(* CODESYS project sfm MES Communication.project

Project tree, tasks and I/O mapping:
  Device : CODESYS Control for Raspberry Pi, 3S - Smart Software Solutions GmbH, version 3.5.11.20
    application Application
      libraries: Standard, * (System); Network, 3.5.7.0 (3S - Smart Software Solutions GmbH); Raspberry I2C Gyroscopes, 1.1.1.0 (3S - Smart Software Solutions GmbH)
      task MainTask (cyclic, interval 4 ms, priority 1) calls PLC_PRG
      task VISU_TASK (cyclic, interval 100 ms, priority 31) calls VisuElems.Visu_Prg
      program PLC_PRG [CFC]
      visualisation Visualization
      function block GetMessage [ST]
      data type Request
      data type Response
      function block TestMES [ST]
    SoftMotion General Axis Pool
    I²C
    SPI
    GPIOs_A_B : GPIOs A/B, 3S - Smart Software Solutions GmbH, version 3.5.11.0
        unmapped channels: digital inputs (GPIO0..GPIO31), digital outputs (GPIO0..GPIO31)
    Onewire
    Camera device
      <Leer>
  text list GlobalTextList
*)

// Device/Application/Request
TYPE Request:
STRUCT
	methodId: INT;
	clientId: INT;
	parameter: INT;
END_STRUCT
END_TYPE

// Device/Application/Response
TYPE Response :
STRUCT
	returnCode: INT;
	para1: INT;
	para2: INT;
END_STRUCT
END_TYPE

// Device/Application/PLC_PRG
PROGRAM PLC_PRG
VAR
	TestMES_0: TestMES;
	GetMessage_0: GetMessage;
	startRequest: BOOL;
	returnCode: INT;
	outPara1: INT;
	outPara2: INT;
	methodId: INT := 400;
	clientId: INT := 1;
	inPara: INT := 0;
	done: BOOL;
END_VAR

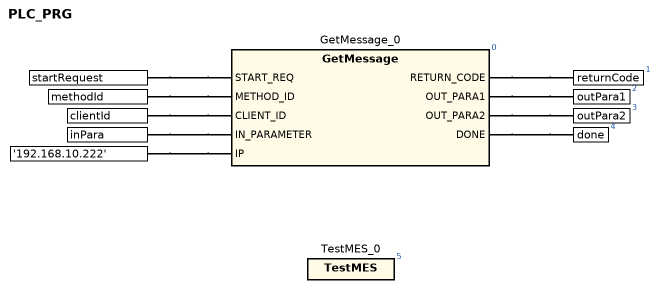
GetMessage_0(
    START_REQ := startRequest,
    METHOD_ID := methodId,
    CLIENT_ID := clientId,
    IN_PARAMETER := inPara,
    IP := '192.168.10.222'); // GetMessage
returnCode := GetMessage_0.RETURN_CODE;
outPara1 := GetMessage_0.OUT_PARA1;
outPara2 := GetMessage_0.OUT_PARA2;
done := GetMessage_0.DONE;
TestMES_0(); // TestMES

END_PROGRAM

// Device/Application/GetMessage
FUNCTION_BLOCK GetMessage
VAR_INPUT
	START_REQ: BOOL;
	METHOD_ID: INT;
	CLIENT_ID: INT;
	IN_PARAMETER: INT;
	IP: STRING;
END_VAR
VAR_OUTPUT
	RETURN_CODE: INT;
	OUT_PARA1: INT;
	OUT_PARA2: INT;
	DONE: BOOL;
END_VAR
VAR
	R_TRIG_StartRequest: R_TRIG;
	request: Request;
	response: Response;
	remotePort: UINT := 2018;
	tcpClient: nbs.TCP_Client;
	tcpWrite: nbs.TCP_Write;
	tcpRead: nbs.TCP_Read;
	targetAddr: NBS.IP_ADDR;
	iStep: INT := 0;
END_VAR


DONE := FALSE;

// wait for rising trigger on input
R_TRIG_StartRequest(CLK:=START_REQ);
IF R_TRIG_StartRequest.Q THEN
	iStep := 10;
END_IF;


CASE iStep OF

	0: 

	10:
		// create connection to server
		DONE := FALSE;
		targetAddr.sAddr := IP;
		tcpClient(xEnable:=TRUE, ipAddr:=targetAddr, uiPort:=remotePort);
		IF tcpClient.xActive THEN
			iStep := 20;  
		END_IF 
		
	20:
		// set values for sending, swap bytes because MES uses different endianess!
		request.methodId := ROL(METHOD_ID, 8);
        request.clientId := ROL(CLIENT_ID, 8);
		request.parameter := ROL(IN_PARAMETER, 8);
		// write to opened connection
		tcpWrite(hConnection:=tcpClient.hConnection, xExecute:=TRUE, pData:=ADR(request), szSize:=SIZEOF(request));
		IF tcpWrite.xDone THEN
			tcpWrite(xExecute:=FALSE);
			iStep := 30;
		END_IF

	30:
		// wait for an answer and read to struct
		tcpRead(hConnection:=tcpClient.hConnection, xEnable:=tcpClient.xActive, pData:=ADR(response), szSize:=SIZEOF(response));	
		IF tcpRead.xReady THEN
			iStep := 40;
		END_IF

	40:
		// set values that were received, swap bytes because MES uses different endianess!
		RETURN_CODE := ROL(Response.returnCode, 8);
		OUT_PARA1 := ROL(Response.para1, 8);
		OUT_PARA2 := ROL(Response.para2, 8);
		DONE := TRUE;

		// close connection
		tcpRead(xEnable:=FALSE);
		tcpClient(xEnable:=FALSE);
		iStep := 0;

END_CASE

END_FUNCTION_BLOCK

// Device/Application/TestMES
FUNCTION_BLOCK TestMES
VAR_INPUT
END_VAR
VAR_OUTPUT
END_VAR
VAR
	getMessage: GetMessage;
	iStep: INT := 0;
END_VAR


// set IP address of MES system
getMessage(ip:='192.168.10.222');

CASE iStep OF
	
	0:
		iStep := 10;
	
	10:
		// startOrder
		getMessage(START_REQ:=TRUE, METHOD_ID:=400, CLIENT_ID:=1, IN_PARAMETER:=0);
		IF getMessage.DONE AND NOT (getMessage.RETURN_CODE = 0) THEN
			getMessage(START_REQ:=FALSE);
			iStep := 20;
		END_IF
		
	20: 
		// startProcess
		getMessage(START_REQ:=TRUE, METHOD_ID:=200, CLIENT_ID:=1, IN_PARAMETER:=0);
		IF getMessage.DONE THEN
			getMessage(START_REQ:=FALSE);
			iStep := 30;
		END_IF
	
	30:
		// endProcess
		getMessage(START_REQ:=TRUE, METHOD_ID:=300, CLIENT_ID:=1, IN_PARAMETER:=0);
		IF getMessage.DONE THEN
			getMessage(START_REQ:=FALSE);
			iStep := 40;
		END_IF
		
	40: 
	
	
END_CASE

END_FUNCTION_BLOCK

// Device/Application/Visualization
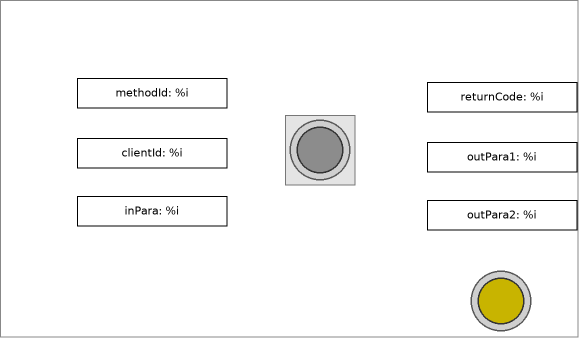
VISUALIZATION Visualization  // 579x338
    PushSwitch (285,115 70x70), variable: PLC_PRG.startRequest, behaviour: TAP, style: Switch-PushSwitch-Gray
    Rectangle (427,82 150x30), "returnCode: %i", text variable: PLC_PRG.returnCode
    Rectangle (427,142 150x30), "outPara1: %i", text variable: PLC_PRG.outPara1
    Rectangle (427,200 150x30), "outPara2: %i", text variable: PLC_PRG.outPara2
    Rectangle (77,78 150x30), "methodId: %i", text variable: PLC_PRG.methodId
    Rectangle (77,138 150x30), "clientId: %i", text variable: PLC_PRG.clientId
    Rectangle (77,196 150x30), "inPara: %i", text variable: PLC_PRG.inPara
    Lamp1 (466,266 70x70), variable: PLC_PRG.done, style: Lamp-Lamp1-Yellow
END_VISUALIZATION
